(* IEC 61131-3 sources: heating/Heating/src, 6 files *)

(* ---- types.iecst ---- *)
TYPE
  SensorsData : STRUCT
    temp1 : INT;         (* keine Initialisierung *)
    temp2 : INT;
  END_STRUCT;
  ActuatorsData : STRUCT
  	valve1 : INT;
  	valve2 : INT;
  END_STRUCT;
END_TYPE

(* ---- input.iecst ---- *)
FUNCTION_BLOCK ReadSensorData
	VAR_INPUT
		p_sensors : REF_TO SensorsData;
	END_VAR

	VAR
		data : REF_TO SensorsData; /* workaround */
	END_VAR

	data := p_sensors; /* workaround */

	/* read data from I/O sub-systems */
END_FUNCTION_BLOCK

(* ---- output.iecst ---- *)
FUNCTION_BLOCK WriteActuators
	VAR_INPUT
		p_actuators : REF_TO ActuatorsData;
	END_VAR

	VAR
		output1 : INT;
	END_VAR

	output1 := p_actuators^.valve1;
END_FUNCTION_BLOCK

(* ---- read_inputs.iecst ---- *)
FUNCTION_BLOCK ReadSensorData
	VAR_INPUT
		p_sensors : REF_TO SensorsData;
	END_VAR

	VAR
		data : REF_TO SensorsData; /* workaround */
		fd : DINT := -1;
		analog_in_1 : ARRAY[0..4] OF UINT;
		digital_in_1 : ARRAY[0..7] OF BOOL;
	END_VAR

	data := p_sensors; /* workaround */

	/* read data from I/O sub-systems */
	IF fd < 0 THEN
		fd := I2C_Open(bus_id := 1); /* /dev/i2c-1 */
	END_IF;

	IF fd >= 0 THEN
		analog_in_1 := I2HAE(fd := fd, address := 16#08);
		data^.ai1 := analog_in_1[0];
		data^.ai2 := analog_in_1[1];
		data^.ai3 := analog_in_1[2];
		data^.ai4 := analog_in_1[3];
		data^.ai5 := analog_in_1[4];

		digital_in_1 := I2C_PCF8574_read(fd := fd, address := 16#20);
		data^.di1 := digital_in_1[0];
		data^.di2 := digital_in_1[1];
		data^.di3 := digital_in_1[2];
		data^.di4 := digital_in_1[3];
		data^.di5 := digital_in_1[4];
		data^.di6 := digital_in_1[5];
		data^.di7 := digital_in_1[6];
		data^.di8 := digital_in_1[7];

		ENO := TRUE;
	ELSE
		ENO := FALSE; /* fd < 0 */
	END_IF;

END_FUNCTION_BLOCK

(* ---- write_outputs.iecst ---- *)
FUNCTION_BLOCK WriteActuators
	VAR_INPUT
		p_actuators : REF_TO ActuatorsData;
	END_VAR

	VAR
		fd : DINT := -1;
		cumm_do_1 : ARRAY[0..7] OF BOOL; /* cumulated digital outputs */
	END_VAR

	ENO := FALSE;

	IF fd < 0 THEN
		fd := I2C_open(bus_id := 1);
	END_IF;

	IF fd >= 0 THEN
		I2HAA(fd := fd, address := 16#58, channel := 0, value := p_actuators^.ao1);
		I2HAA(fd := fd, address := 16#58, channel := 1, value := p_actuators^.ao2);
		I2HAA(fd := fd, address := 16#58, channel := 2, value := p_actuators^.ao3);
		I2HAA(fd := fd, address := 16#58, channel := 3, value := p_actuators^.ao4);

		cumm_do_1[0] := p_actuators^.do1;
		cumm_do_1[1] := p_actuators^.do2;
		cumm_do_1[2] := p_actuators^.do3;
		cumm_do_1[3] := p_actuators^.do4;
		cumm_do_1[4] := p_actuators^.do5;
		cumm_do_1[5] := p_actuators^.do6;
		cumm_do_1[6] := p_actuators^.do7;
		cumm_do_1[7] := p_actuators^.do8;
		I2C_PCF8574_write(fd := fd, address := 16#38, pin_values := cumm_do_1);
		ENO := TRUE;
	ELSE
		ENO := FALSE;
	END_IF;

END_FUNCTION_BLOCK

(* ---- main.iecst ---- *)
PROGRAM Heating
	VAR
		/* I/O image */
		sensors : SensorsData;
		actuators : ActuatorsData;

		/* I/O access functions */
		read : ReadSensorData;
		write : WriteActuators;
	END_VAR

	read(p_sensors := REF(sensors));

	actuators.valve1 := sensors.temp1 * 2; /* example of controller logic */

	write(p_actuators := REF(actuators));

END_PROGRAM
